FUNCTION_BLOCK WP_SENSE (* Workpiece presence and style sensor *)
  (* Standard: 61499-1; Classification: Simulation *)
  (* Version 0.2, 2005-06-01, JHC, Holobloc Inc, Re-compiled with new emitter. *)
  (* Version 0.1, 2002-04-20, JHC, Rockwell Automation, Moved to fb.rt.mva *)
  (* Version 0.0, 2002-04-10, JHC, Rockwell Automation *)
  (* Compiler header: package fb.rt.mva; *)
  (* Compiler Java IBM VisualAge 3.0 *)
  (* Compiler Java IBM Jikes 1.06 *)
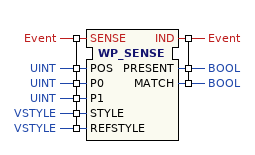
  EVENT_INPUT
    SENSE WITH STYLE, REFSTYLE, POS, P0, P1; (* Input change notification *)
  END_EVENT
  EVENT_OUTPUT
    IND WITH PRESENT, MATCH; (* Output change indication *)
  END_EVENT
  VAR_INPUT
    POS : UINT; (* Workpiece position on conveyor (0-100%) *)
    P0 : UINT; (* Position sensor lower limit *)
    P1 : UINT; (* Position sensor upper limit *)
    STYLE : VSTYLE; (* Workpiece style *)
    REFSTYLE : VSTYLE; (* Style to be sensed *)
  END_VAR
  VAR_OUTPUT
    PRESENT : BOOL; (* Workpiece is present between P0 and P1 *)
    MATCH : BOOL; (* Workpiece is present and STYLE matches REFSTYLE *)
  END_VAR
  ALGORITHM SENSE IN Java:
boolean newpres = (POS.value>=P0.value)&&(POS.value<=P1.value)&&(STYLE.value != VSTYLE.NONE);
boolean newmatch = newpres & (STYLE.equals(REFSTYLE));
if((newpres != PRESENT.value)||(newmatch != MATCH.value)){
   PRESENT.value = newpres;
   MATCH.value = newmatch;
   IND.serviceEvent(this);}
  END_ALGORITHM
END_FUNCTION_BLOCK
